TYPE DUT_PneumaticActuator_Position :
(RETRACTED, INSERTED, MOVING, INVALID);
END_TYPE

(* stored: Version 1.1.0.1, ProductVersion 3.1.4022.18
   DUT DUT_PneumaticActuator_Position: Id {61a5e714-50c7-4f12-a7ea-a0cbcc21a898} *)
